FUNCTION_BLOCK FB_Test
VAR_INPUT

END_VAR
VAR_OUTPUT
END_VAR
VAR
	j : INT;
	fbTest2 : FB_Test2;
END_VAR

PROPERTY PUBLIC Prop : INT
GET
Prop := j;
END_GET
END_PROPERTY

END_FUNCTION_BLOCK

(* stored: Version 1.1.0.1, ProductVersion 3.1.4024.12
   POU FB_Test: Id {0d004d85-cf62-4d44-ab7f-7558084e159f}, SpecialFunc None
   Property Prop: Id {cc5b34cf-ed59-4797-9329-a4ac54e5d15d}
   Get Get: Id {8e6dc78c-b80a-4229-bec9-d09633b3d81f} *)
